TYPE ST_PML_Base_Out :
STRUCT
	eStateCurrent		: E_PackMLState := E_PackMLState.Undefined;
	eStatePrevious		: E_PackMLState := E_PackMLState.Undefined;
	eModeCurrent		: T_PackMLMode := E_PackMLMode.Unknown;
	eModePrevious		: T_PackMLMode := E_PackMLMode.Unknown;

	bCommandAccepted	: BOOL;
	bCommandRejected	: BOOL;
	eStateErrorID		: E_PackMLErrorID := E_PackMLErrorID.NoError;

	bModeChanged		: BOOL;
	bModeChangeRejected	: BOOL;
	eModeErrorID		: E_PackMLErrorID := E_PackMLErrorID.NoError;
END_STRUCT
END_TYPE

(* stored: Version 1.1.0.1, ProductVersion 3.1.4026.18
   DUT ST_PML_Base_Out: Id {ebcaecfd-ea1d-45e9-b675-b2f07f9d66c3} *)
